PROGRAM MAIN
VAR
END_VAR

END_PROGRAM

(* stored: Version 1.1.0.1, ProductVersion 3.1.4024.11
   POU MAIN: Id {02ad2c29-6642-49c8-88da-ed2d175dbf50}, SpecialFunc None *)
